FUNCTION_BLOCK PUBL_1 (* Single-Variable Local Group Publisher *)
  (* Standard: 61499-1; Classification: Communications *)
  (* Version 0.1, 2002-05-02, JHC, Rockwell Automation, Optimized. *)
  (* Version 0.0, 2001-10-02, JHC, Rockwell Automation, Copied/modified from PUBLISH_1 *)
  (* Compiler header: package fb.rt.net; *)
  (* Compiler Java IBM VisualAge 3.0 *)
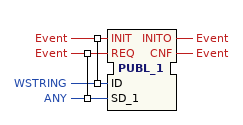
  EVENT_INPUT
    INIT WITH ID; (* Service Initialization *)
    REQ WITH SD_1; (* Service Request *)
  END_EVENT
  EVENT_OUTPUT
    INITO; (* Initialization Confirm *)
    CNF; (* Service Confirmation *)
  END_EVENT
  VAR_INPUT
    ID : WSTRING; (* Local Group Name-Default is FB Instance Name *)
    SD_1 : ANY; (* Data to Send *)
  END_VAR
  SERVICE PUBL_1/SUBL_1 (* Data Publication Service *)
    SEQUENCE normal_establishment
      PUBL_1.INIT(ID) -> PUBL_1.INITO();
      SUBL_1.INIT(ID) -> SUBL_1.INITO();
    END_SEQUENCE
    SEQUENCE normal_data_transfer
      PUBL_1.REQ(SD_1) -> SUBL_1.IND(RD_1) -> PUBL_1.CNF();
    END_SEQUENCE
  END_SERVICE
END_FUNCTION_BLOCK
